# EPICS substitutions: db/EL1012.substitutions
file EL1012.template
{ 	pattern
	{
		TERMINAL,
		DESC1,	ZNAM1,	ONAM1,	ZSV1,	OSV1,	COSV1,	SCAN1,
		DESC2,	ZNAM2,	ONAM2,	ZSV2,	OSV2,	COSV2,	SCAN2
	}
	{
	}
}
